{attribute 'hide_all_locals'}
FUNCTION_BLOCK PUBLIC FB_FullTimeEmployee EXTENDS FB_Employee
VAR_INPUT
END_VAR
VAR_OUTPUT
END_VAR
VAR
	nAnnualSalaryBacking	:	UINT;
END_VAR

METHOD PUBLIC GetMonthlySalary : LREAL
VAR_INPUT
END_VAR
GetMonthlySalary := nAnnualSalary / 12;
END_METHOD

{attribute 'monitoring' := 'variable'}
PROPERTY PUBLIC nAnnualSalary : UINT
GET
nAnnualSalary := nAnnualSalaryBacking;
END_GET
SET
nAnnualSalaryBacking := nAnnualSalary;
END_SET
END_PROPERTY

END_FUNCTION_BLOCK

(* stored: Version 1.1.0.1, ProductVersion 3.1.4024.12
   POU FB_FullTimeEmployee: Id {a3fcde26-925a-40bc-9c5d-c909b2dc2c4f}, SpecialFunc None
   Method GetMonthlySalary: Id {19b65e9d-1ce3-41b1-864d-5a175dc14c55}
   Property nAnnualSalary: Id {ecc488aa-1029-4a23-bad9-42ea4e1652f0}
   Get Get: Id {f7edb5cb-5589-45d3-ae3a-a93f8aec8744}
   Set Set: Id {8cae3932-cb3a-4432-9437-9675c2091110} *)
